// TIA Portal V19 export
ORGANIZATION_BLOCK "Main"   // OB1, LAD, ProgramCycle
TITLE = "Main Program Sweep (Cycle)"
{ S7_Optimized_Access := 'TRUE' }
// stored: SetENOAutomatically false
   VAR_INPUT
      Initial_Call : Bool;   // Initial call of this OB
      Remanence : Bool;   // =True, if remanent data are available
   END_VAR
   VAR_TEMP   // added for the SCL form of the ladder/FBD networks
      _w1 : Bool;
   END_VAR
BEGIN

REGION Network 1
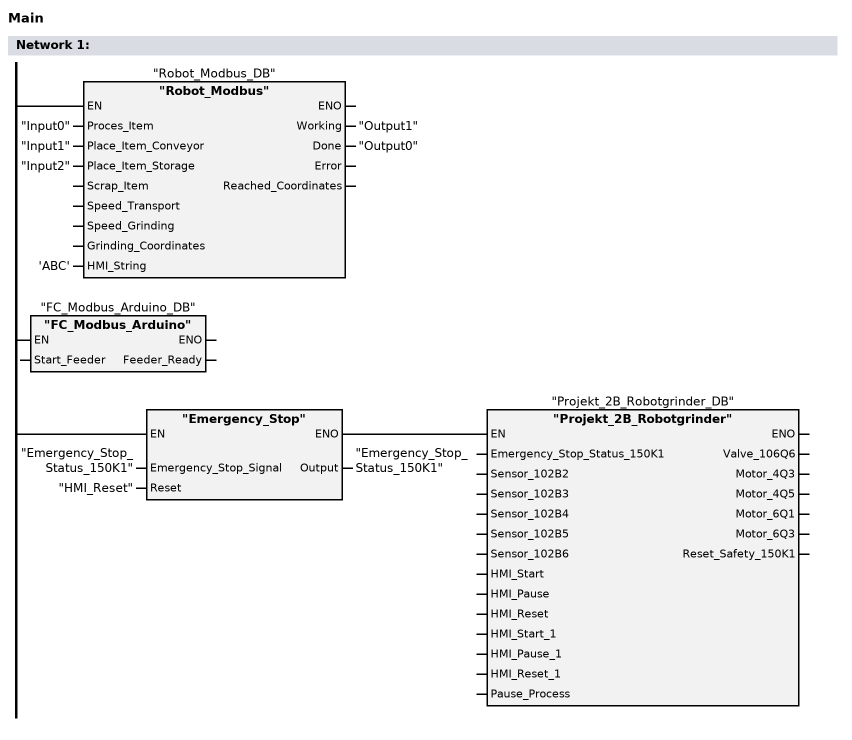
   RUNG wire#powerrail
      "Robot_Modbus_DB"(Proces_Item := "Input0", Place_Item_Conveyor := "Input1", Place_Item_Storage := "Input2", Scrap_Item :=, Speed_Transport :=, Speed_Grinding :=, Grinding_Coordinates :=, HMI_String := 'ABC', Working => "Output1", Done => "Output0", Error =>, Reached_Coordinates =>)
   END_RUNG
   RUNG wire#powerrail
      "FC_Modbus_Arduino_DB"(Start_Feeder :=, Feeder_Ready =>)
   END_RUNG
   RUNG wire#powerrail
      "Emergency_Stop"(Emergency_Stop_Signal := "Emergency_Stop_Status_150K1", Reset := "HMI_Reset", Output => "Emergency_Stop_Status_150K1")
      "Projekt_2B_Robotgrinder_DB"(Emergency_Stop_Status_150K1 :=, Sensor_102B2 :=, Sensor_102B3 :=, Sensor_102B4 :=, Sensor_102B5 :=, Sensor_102B6 :=, HMI_Start :=, HMI_Pause :=, HMI_Reset :=, HMI_Start_1 :=, HMI_Pause_1 :=, HMI_Reset_1 :=, Pause_Process :=, Valve_106Q6 =>, Motor_4Q3 =>, Motor_4Q5 =>, Motor_6Q1 =>, Motor_6Q3 =>, Reset_Safety_150K1 =>)
   END_RUNG
   // the same network as SCL:
   "Robot_Modbus_DB"(Proces_Item := "Input0",   // "Robot_Modbus"
                     Place_Item_Conveyor := "Input1",
                     Place_Item_Storage := "Input2",
                     HMI_String := 'ABC',
                     Working => "Output1",
                     Done => "Output0");
   "FC_Modbus_Arduino_DB"();   // "FC_Modbus_Arduino"
   "Emergency_Stop"(Emergency_Stop_Signal := "Emergency_Stop_Status_150K1",
                    Reset := "HMI_Reset",
                    Output => "Emergency_Stop_Status_150K1",
                    ENO => #_w1);
   IF #_w1 THEN
       "Projekt_2B_Robotgrinder_DB"();   // "Projekt_2B_Robotgrinder"
   END_IF;
END_REGION
END_ORGANIZATION_BLOCK
